FUNCTION_BLOCK FB_BWK_Ablaufsteuerung
VAR_IN_OUT
	Zustand			: ST_BWK_Zustand;
	Stellwert			: ST_BWK_Stellwert;
END_VAR
VAR_INPUT
	Steuerung		: ST_BWK_Steuerung;
	Parameter		: ST_BWK_Parameter;
END_VAR
VAR_OUTPUT
END_VAR
VAR
	Timer			: TON;
END_VAR

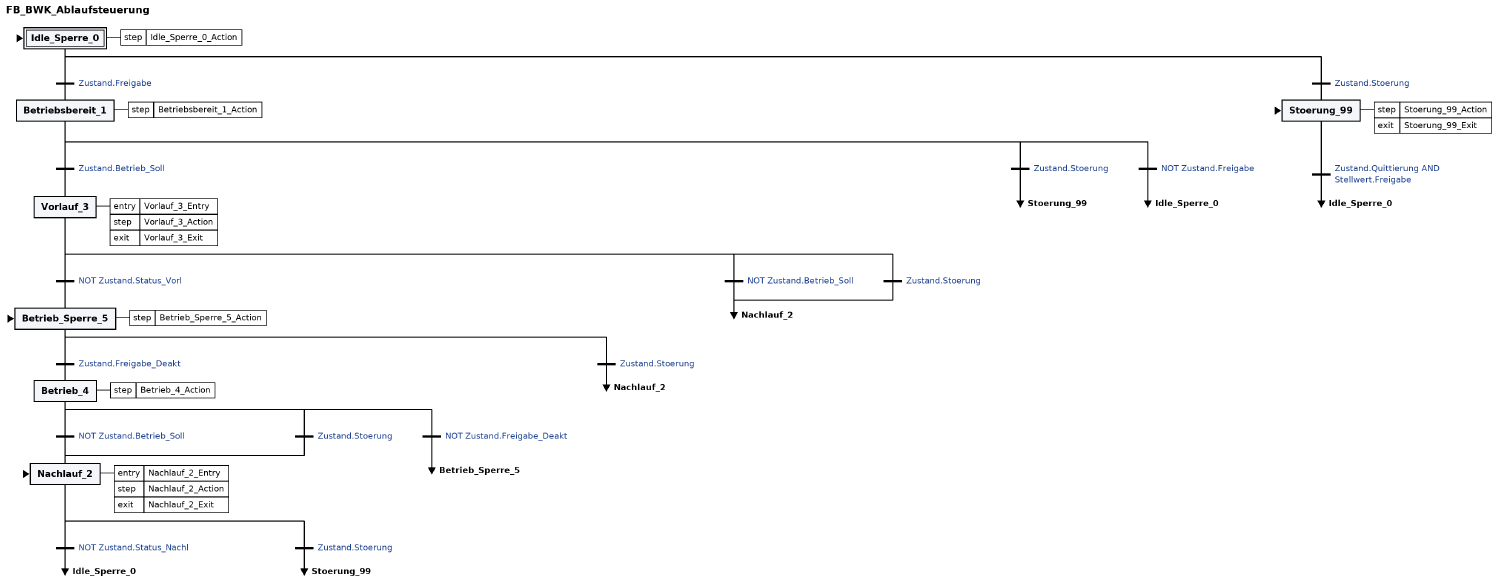
INITIAL_STEP Idle_Sperre_0:
    Idle_Sperre_0_Action(N);  // step action
END_STEP
TRANSITION FROM Idle_Sperre_0 TO Betriebsbereit_1
    := Zustand.Freigabe;
END_TRANSITION
TRANSITION FROM Idle_Sperre_0 TO Stoerung_99
    := Zustand.Stoerung;
END_TRANSITION
STEP Stoerung_99:
    Stoerung_99_Action(N);  // step action
    Stoerung_99_Exit(P0);  // exit action
END_STEP
TRANSITION FROM Stoerung_99 TO Idle_Sperre_0
    := Zustand.Quittierung AND Stellwert.Freigabe;
END_TRANSITION
STEP Betriebsbereit_1:
    Betriebsbereit_1_Action(N);  // step action
END_STEP
TRANSITION FROM Betriebsbereit_1 TO Vorlauf_3
    := Zustand.Betrieb_Soll;
END_TRANSITION
TRANSITION FROM Betriebsbereit_1 TO Stoerung_99
    := Zustand.Stoerung;
END_TRANSITION
TRANSITION FROM Betriebsbereit_1 TO Idle_Sperre_0
    := NOT Zustand.Freigabe;
END_TRANSITION
STEP Vorlauf_3:
    Vorlauf_3_Entry(P1);  // entry action
    Vorlauf_3_Action(N);  // step action
    Vorlauf_3_Exit(P0);  // exit action
END_STEP
TRANSITION FROM Vorlauf_3 TO Betrieb_Sperre_5
    := NOT Zustand.Status_Vorl;
END_TRANSITION
TRANSITION FROM Vorlauf_3 TO Nachlauf_2
    := NOT Zustand.Betrieb_Soll;
END_TRANSITION
TRANSITION FROM Vorlauf_3 TO Nachlauf_2
    := Zustand.Stoerung;
END_TRANSITION
STEP Betrieb_Sperre_5:
    Betrieb_Sperre_5_Action(N);  // step action
END_STEP
TRANSITION FROM Betrieb_Sperre_5 TO Betrieb_4
    := Zustand.Freigabe_Deakt;
END_TRANSITION
TRANSITION FROM Betrieb_Sperre_5 TO Nachlauf_2
    := Zustand.Stoerung;
END_TRANSITION
STEP Betrieb_4:
    Betrieb_4_Action(N);  // step action
END_STEP
TRANSITION FROM Betrieb_4 TO Nachlauf_2
    := NOT Zustand.Betrieb_Soll;
END_TRANSITION
TRANSITION FROM Betrieb_4 TO Nachlauf_2
    := Zustand.Stoerung;
END_TRANSITION
TRANSITION FROM Betrieb_4 TO Betrieb_Sperre_5
    := NOT Zustand.Freigabe_Deakt;
END_TRANSITION
STEP Nachlauf_2:
    Nachlauf_2_Entry(P1);  // entry action
    Nachlauf_2_Action(N);  // step action
    Nachlauf_2_Exit(P0);  // exit action
END_STEP
TRANSITION FROM Nachlauf_2 TO Idle_Sperre_0
    := NOT Zustand.Status_Nachl;
END_TRANSITION
TRANSITION FROM Nachlauf_2 TO Stoerung_99
    := Zustand.Stoerung;
END_TRANSITION

ACTION Betrieb_4_Action:
(* Stellwert setzen *)
Stellwert.Betrieb := TRUE;

(* Zustand setzen *)
Zustand.Status := E_BWK_Zustand_Status_Betrieb;
END_ACTION

ACTION Betrieb_Sperre_5_Action:
(* Stellwert setzen *)
Stellwert.Betrieb := TRUE;

(* Zustand setzen *)
Zustand.Status := E_BWK_Zustand_Status_Betrieb_Sperre;
END_ACTION

ACTION Betriebsbereit_1_Action:
(* Stellwert setzen *)
Stellwert.Betrieb := FALSE;
Stellwert.Freigabe := TRUE;

(* Zustand setzen *)
Zustand.Status := E_BWK_Zustand_Status_Betriebsbereit;
END_ACTION

ACTION Idle_Sperre_0_Action:
(* Stellwert setzen *)
Stellwert.Betrieb := FALSE;

(* Zustand setzen *)
Zustand.Status := E_BWK_Zustand_Status_Idle_Sperre;
END_ACTION

ACTION Nachlauf_2_Action:
(* Nachlauf Timer starten *)
Timer( 	IN := Zustand.Status_Nachl,
		PT := DINT_TO_TIME(Parameter.Zeit_Nachl)
);
Zustand.Status_Nachl	:= NOT(Timer.Q AND NOT Zustand.Betrieb);

(* Stellwert setzen *)
Stellwert.Betrieb := FALSE;
Stellwert.Freigabe := FALSE;

(* Zustand setzen *)
Zustand.Status := E_BWK_Zustand_Status_Nachl;
END_ACTION

ACTION Nachlauf_2_Entry:
Zustand.Status_Nachl := TRUE;
(* Reset Timer *)
Timer(IN := FALSE);
END_ACTION

ACTION Nachlauf_2_Exit:
Zustand.Status_Nachl := FALSE;
END_ACTION

ACTION Stoerung_99_Action:
(* Stellwert setzen *)
Stellwert.Betrieb := FALSE;

(* Zustand setzen *)
Zustand.Stoerung := TRUE;
Zustand.Status := E_BWK_Zustand_Status_Stoerung;
END_ACTION

ACTION Stoerung_99_Exit:
Zustand.Stoerung	:= FALSE;
END_ACTION

ACTION Vorlauf_3_Action:
(* Vorlaufzeit Timer starten *)
Timer( 	IN := Zustand.Status_Vorl,
		PT := DINT_TO_TIME(Parameter.Zeit_Vorl)
);
Zustand.Status_Vorl := NOT (Timer.Q AND Zustand.Betrieb);

(* Stellwert setzen *)
IF Stellwert.Freigabe THEN
	Stellwert.Betrieb := TRUE;
END_IF

(* Zustand setzen *)
Zustand.Status := E_BWK_Zustand_Status_Vorl;
END_ACTION

ACTION Vorlauf_3_Entry:
Zustand.Status_Vorl := TRUE;
(* Reset Timer *)
Timer(IN := FALSE);
END_ACTION

ACTION Vorlauf_3_Exit:
Zustand.Status_Vorl := FALSE;
END_ACTION

END_FUNCTION_BLOCK

(* stored: Version 1.1.0.1, ProductVersion 3.1.4024.9
   POU FB_BWK_Ablaufsteuerung: Id {ab81f34c-e313-4323-b276-469a25746313}, SpecialFunc None
   Action Betrieb_4_Action: Id {1e9859dc-b629-46e8-9624-d68831898fb2}
   Action Betrieb_Sperre_5_Action: Id {6c6784c6-b188-44e8-901e-934a79641717}
   Action Betriebsbereit_1_Action: Id {e2bde419-11c1-47ac-889a-5f3a11ec9b9a}
   Action Idle_Sperre_0_Action: Id {1912f694-fc63-4150-b13b-14a6f66e04c3}
   Action Nachlauf_2_Action: Id {88256271-139c-4623-9fba-777ae91c7ffb}
   Action Nachlauf_2_Entry: Id {645f9918-a9a1-4cc0-b384-344f07c34624}
   Action Nachlauf_2_Exit: Id {2b125d2c-56ae-48a5-846c-5fdf7fd32e6b}
   Action Stoerung_99_Action: Id {9ba06089-ac34-4f17-b9bb-5d3c69570868}
   Action Stoerung_99_Exit: Id {2a64c0fb-acde-4911-a345-cbe9391a5bc8}
   Action Vorlauf_3_Action: Id {46ca5131-daa6-42d8-bc27-6820c7d11d44}
   Action Vorlauf_3_Entry: Id {dc5641de-6b68-4c8f-88a7-4145e14a7e55}
   Action Vorlauf_3_Exit: Id {b50a9c5d-03b7-4a89-9fcb-79ada70fb4dd} *)
